NETWORK
TITLE = ---- Accion del Evento --> Peticion de Refresco del Dispositivo Barrera
///////////////////////////////////////////////////////////////////////////////
///////////////////////////////////////////////////////////////////////////////
///////////////////////////////////////////////////////////////////////////////
// Dispositivos tipo Barrera uno determinado o todos
DispositivoBarrera_EventoRecibido_RefrescoDispositivo:NOP   0;
      SET;
      L     #AtributosDeDispositivos.Numero;  // Mirar si hay numero de maquina
      L     0;  // Son todos las Barreras
      ==I;
      JC    DispositivosTodosBarrera_EventoRecibido_RefrescoDispositivo;


///////////////////////////////////////////////////////////////////////////////
// --- Es Una Maquina Determinada
      JU    DispositivosUnaBarrera_EventoRecibido_RefrescoDispositivo;



NETWORK
TITLE = ---- ---- De una Barrera
///////////////////////////////////////////////////////////////////////////////
///////////////////////////////////////////////////////////////////////////////
///////////////////////////////////////////////////////////////////////////////
// --- Una Barrera  determinada
DispositivosUnaBarrera_EventoRecibido_RefrescoDispositivo:NOP   0;

      L     #AtributosDeDispositivos.Numero;  // Ver que Barrera es
      L     "CTE_OffsetMesa";
      -I;
      T     #VarTempDispositivos.Numero;

      L     #VarTempDispositivos.Numero;  // Comprobar el numero de Barrera
      L     1;  // No menor de 1
      <I;  // No es correcto
      JC    Final_EventoRecibido_RefrescoDispositivo;
      L     #VarTempDispositivos.Numero;
      L     "CTE_MaxDispositivosBarrera";  // No meyor que el parametro
      >I;  // No es correcto
      JC    Final_EventoRecibido_RefrescoDispositivo;


///////////////////////////////////////////////////////////////////////////////
// --- Activar Refresco del Dispositivo
///////////////////////////////////////////////////////////////////////////////
// Activar Refresco del Dispositivo
      SET;
      S     "DB839_DispositivosVarios".DispoBarrera[#VarTempDispositivos.Numero].RefrescoDatos;


///////////////////////////////////////////////////////////////////////////////
// --- Finalizar
      JU    Final_EventoRecibido_RefrescoDispositivo;



NETWORK
TITLE = ---- ---- De Todas las Barreras
////////////////////////////////////////////////////////////////////////////
////////////////////////////////////////////////////////////////////////////
////////////////////////////////////////////////////////////////////////////
// --- Peticion de Todos los dispositivos BARRERA
DispositivosTodosBarrera_EventoRecibido_RefrescoDispositivo:NOP   0;
      L     1;
      T     #IndiceDispositivosVarios;


////////////////////////////////////////////////////////////////////////////
////////////////////////////////////////////////////////////////////////////
////////////////////////////////////////////////////////////////////////////
BucleBarrera_EventoRecibido_RefrescoDispositivo:NOP   0;


///////////////////////////////////////////////////////////////////////////////
// Activar Refresco del Dispositivo
      SET;
      S     "DB839_DispositivosVarios".DispoBarrera[#IndiceDispositivosVarios].RefrescoDatos;
////////////////////////////////////////////////////////////////////////////
      L     #IndiceDispositivosVarios;  // Siguiente Dispositivo
      L     1;
      +I;
      T     #IndiceDispositivosVarios;

      L     #IndiceDispositivosVarios;
      L     "CTE_MaxDispositivosBarrera";
      >I;  // Ha superado el maximo ??
      JC    FinBucleBarrera_EventoRecibido_RefrescoDispositivo;

      JU    BucleBarrera_EventoRecibido_RefrescoDispositivo;  // Continuar en el Bucle


////////////////////////////////////////////////////////////////////////////
////////////////////////////////////////////////////////////////////////////
////////////////////////////////////////////////////////////////////////////
FinBucleBarrera_EventoRecibido_RefrescoDispositivo:NOP   0;
      JU    Final_EventoRecibido_RefrescoDispositivo;


NETWORK
TITLE = ---- Accion del Evento --> Peticion de Refresco del Dispositivo Puerta
///////////////////////////////////////////////////////////////////////////////
///////////////////////////////////////////////////////////////////////////////
///////////////////////////////////////////////////////////////////////////////
// Dispositivos tipo Puerta uno determinado o todos
DispositivoPuerta_EventoRecibido_RefrescoDispositivo:NOP   0;
      SET;
      L     #AtributosDeDispositivos.Numero;  // Mirar si hay numero de maquina
      L     0;  // Son todos las Puertas
      ==I;
      JC    DispositivosTodosPuerta_EventoRecibido_RefrescoDispositivo;


///////////////////////////////////////////////////////////////////////////////
// --- Es Una Maquina Determinada
      JU    DispositivosUnaPuerta_EventoRecibido_RefrescoDispositivo;



NETWORK
TITLE = ---- ---- De una Puerta
///////////////////////////////////////////////////////////////////////////////
///////////////////////////////////////////////////////////////////////////////
///////////////////////////////////////////////////////////////////////////////
// --- Uan Puerta determinada
DispositivosUnaPuerta_EventoRecibido_RefrescoDispositivo:NOP   0;

      L     #AtributosDeDispositivos.Numero;  // Ver que Puerta es
      L     "CTE_OffsetMesa";
      -I;
      T     #VarTempDispositivos.Numero;

      L     #VarTempDispositivos.Numero;  // Comprobar el numero de Puerta
      L     1;  // No menor de 1
      <I;  // No es correcto
      JC    Final_EventoRecibido_RefrescoDispositivo;
      L     #VarTempDispositivos.Numero;
      L     "CTE_MaxDispositivosPuerta";  // No meyor que el parametro
      >I;  // No es correcto
      JC    Final_EventoRecibido_RefrescoDispositivo;


///////////////////////////////////////////////////////////////////////////////
// --- Activar Refresco del Dispositivo
///////////////////////////////////////////////////////////////////////////////
// Activar Refresco del Dispositivo
      SET;
      S     "DB839_DispositivosVarios".DispoPuerta[#VarTempDispositivos.Numero].RefrescoDatos;


///////////////////////////////////////////////////////////////////////////////
// --- Finalizar
      JU    Final_EventoRecibido_RefrescoDispositivo;



NETWORK
TITLE = ---- ---- De Todas las Puertas
////////////////////////////////////////////////////////////////////////////
////////////////////////////////////////////////////////////////////////////
////////////////////////////////////////////////////////////////////////////
// --- Peticion de Todos los dispositivos PUERTA
DispositivosTodosPuerta_EventoRecibido_RefrescoDispositivo:NOP   0;
      L     1;
      T     #IndiceDispositivosVarios;


////////////////////////////////////////////////////////////////////////////
////////////////////////////////////////////////////////////////////////////
////////////////////////////////////////////////////////////////////////////
BuclePuerta_EventoRecibido_RefrescoDispositivo:NOP   0;


///////////////////////////////////////////////////////////////////////////////
// Activar Refresco del Dispositivo
      SET;
      S     "DB839_DispositivosVarios".DispoPuerta[#IndiceDispositivosVarios].RefrescoDatos;

////////////////////////////////////////////////////////////////////////////
      L     #IndiceDispositivosVarios;  // Siguiente Dispositivo
      L     1;
      +I;
      T     #IndiceDispositivosVarios;

      L     #IndiceDispositivosVarios;
      L     "CTE_MaxDispositivosPuerta";
      >I;  // Ha superado el maximo ??
      JC    FinBuclePuerta_EventoRecibido_RefrescoDispositivo;

      JU    BuclePuerta_EventoRecibido_RefrescoDispositivo;  // Continuar en el Bucle


////////////////////////////////////////////////////////////////////////////
////////////////////////////////////////////////////////////////////////////
////////////////////////////////////////////////////////////////////////////
FinBuclePuerta_EventoRecibido_RefrescoDispositivo:NOP   0;
      JU    Final_EventoRecibido_RefrescoDispositivo;


NETWORK
TITLE = ---- Accion del Evento --> Peticion de Refresco del Dispositivo Linea de Potencia
///////////////////////////////////////////////////////////////////////////////
///////////////////////////////////////////////////////////////////////////////
///////////////////////////////////////////////////////////////////////////////
// Dispositivos tipo Linea de Potencia uno determinado o todos
DispositivoLineaPotencia_EventoRecibido_RefrescoDispositivo:NOP   0;
      SET;
      L     #AtributosDeDispositivos.Numero;  // Mirar si hay numero de maquina
      L     0;  // Son todos las Lineas de Potencia
      ==I;
      JC    DispositivosTodosLineaPotencia_EventoRecibido_RefrescoDispositivo;


///////////////////////////////////////////////////////////////////////////////
// --- Es Una Maquina Determinada
      JU    DispositivosUnaLineaPotencia_EventoRecibido_RefrescoDispositivo;



NETWORK
TITLE = ---- ---- De una Linea de Potencia
///////////////////////////////////////////////////////////////////////////////
///////////////////////////////////////////////////////////////////////////////
///////////////////////////////////////////////////////////////////////////////
// --- Maquina  determinada
DispositivosUnaLineaPotencia_EventoRecibido_RefrescoDispositivo:NOP   0;

      L     #AtributosDeDispositivos.Numero;  // Ver que Linea de Potencia es
      L     "CTE_OffsetMesa";
      -I;
      T     #VarTempDispositivos.Numero;

      L     #VarTempDispositivos.Numero;  // Comprobar el numero de Linea de Potencia
      L     1;  // No menor de 1
      <I;  // No es correcto
      JC    Final_EventoRecibido_RefrescoDispositivo;
      L     #VarTempDispositivos.Numero;
      L     "CTE_MaxDispositivosLineaPotencia";  // No meyor que el parametro
      >I;  // No es correcto
      JC    Final_EventoRecibido_RefrescoDispositivo;


///////////////////////////////////////////////////////////////////////////////
// --- Activar Refresco del Dispositivo
///////////////////////////////////////////////////////////////////////////////
// Activar Refresco del Dispositivo
      SET;
      S     "DB839_DispositivosVarios".DispoLineaPotencia[#VarTempDispositivos.Numero].RefrescoDatos;


///////////////////////////////////////////////////////////////////////////////
// --- Finalizar
      JU    Final_EventoRecibido_RefrescoDispositivo;



NETWORK
TITLE = ---- ---- De Todas Las Lineas de Potencia
////////////////////////////////////////////////////////////////////////////
////////////////////////////////////////////////////////////////////////////
////////////////////////////////////////////////////////////////////////////
// --- Peticion de Todos los dispositivos LINEA DE POTENCIA
DispositivosTodosLineaPotencia_EventoRecibido_RefrescoDispositivo:NOP   0;
      L     1;
      T     #IndiceDispositivosVarios;


////////////////////////////////////////////////////////////////////////////
////////////////////////////////////////////////////////////////////////////
////////////////////////////////////////////////////////////////////////////
BucleLineaPotencia_EventoRecibido_RefrescoDispositivo:NOP   0;


///////////////////////////////////////////////////////////////////////////////
// Activar Refresco del Dispositivo
      SET;
      S     "DB839_DispositivosVarios".DispoLineaPotencia[#IndiceDispositivosVarios].RefrescoDatos;

////////////////////////////////////////////////////////////////////////////
      L     #IndiceDispositivosVarios;  // Siguiente Dispositivo
      L     1;
      +I;
      T     #IndiceDispositivosVarios;

      L     #IndiceDispositivosVarios;
      L     "CTE_MaxDispositivosLineaPotencia";
      >I;  // Ha superado el maximo ??
      JC    FinBucleLineaPotencia_EventoRecibido_RefrescoDispositivo;

      JU    BucleLineaPotencia_EventoRecibido_RefrescoDispositivo;  // Continuar en el Bucle


////////////////////////////////////////////////////////////////////////////
////////////////////////////////////////////////////////////////////////////
////////////////////////////////////////////////////////////////////////////
FinBucleLineaPotencia_EventoRecibido_RefrescoDispositivo:NOP   0;
      JU    Final_EventoRecibido_RefrescoDispositivo;


NETWORK
TITLE = ---- Accion del Evento --> Peticion de Refresco de Todos Los Dispositivos
///////////////////////////////////////////////////////////////////////////////
///////////////////////////////////////////////////////////////////////////////
///////////////////////////////////////////////////////////////////////////////
// --- Todos los dispositivos
DispositivosTodos_EventoRecibido_RefrescoDispositivo:NOP   0;



NETWORK
TITLE = ---- ---- CCPIF y CBOX
///////////////////////////////////////////////////////////////////////////////
///////////////////////////////////////////////////////////////////////////////
///////////////////////////////////////////////////////////////////////////////
// --- Recorrer CCPIF y Todos los CBOX
      L     0;
      T     #IndiceCBOX;


///////////////////////////////////////////////////////////////////////////////
///////////////////////////////////////////////////////////////////////////////
///////////////////////////////////////////////////////////////////////////////
BucleArmarios_DispositivosTodos_EventoRecibido_RefrescoDispositivo:NOP   0;


///////////////////////////////////////////////////////////////////////////////
/// --- Inicio si pertenece al JDT
      SET;
      X     "DB855_DefinicionDispositivos".Dispositivos[#IndiceCBOX].EventosDelJdT02;
      XN    #JDT02_Activo;
      =     #DispositivoDeJDT02;

      SET;
      AN    #DispositivoDeJDT02;
      JC    ContinuarBucleArmarios_DispositivosTodos_EventoRecibido_RefrescoDispositivo;


///////////////////////////////////////////////////////////////////////////////
// --- Activar Refresco del Dispositivo
      L     250;  // 250 - Recibido Evento de Refresco de Datos del Dispositivo
      T     "DB830_Dispositivos".Dispositivos[#IndiceCBOX].EstadoRecepcionEvento;


///////////////////////////////////////////////////////////////////////////////
ContinuarBucleArmarios_DispositivosTodos_EventoRecibido_RefrescoDispositivo:NOP   0;
      L     #IndiceCBOX;  // Incremento al siguiente CBOX
      L     1;
      +I;
      T     #IndiceCBOX;

      L     #IndiceCBOX;
      L     "CTE_MaxDispositivos";
      >I;  // Finalizar
      JC    FinBucleArmarios_DispositivosTodos_EventoRecibido_RefrescoDispositivos;

///////////////////////////////////////////////////////////////////////////////
// --- Ir hacia el siguiente CBOX
      JU    BucleArmarios_DispositivosTodos_EventoRecibido_RefrescoDispositivo;


///////////////////////////////////////////////////////////////////////////////
///////////////////////////////////////////////////////////////////////////////
///////////////////////////////////////////////////////////////////////////////
FinBucleArmarios_DispositivosTodos_EventoRecibido_RefrescoDispositivos:NOP   0;



NETWORK
TITLE = ---- ---- Mesas
///////////////////////////////////////////////////////////////////////////////
///////////////////////////////////////////////////////////////////////////////
// Recorrer Todas las Mesas
      L     1;
      T     #IndiceMesa;

///////////////////////////////////////////////////////////////////////////////
///////////////////////////////////////////////////////////////////////////////
///////////////////////////////////////////////////////////////////////////////
BucleMesas_DispositivosTodos_EventoRecibido_RefrescoDispositivo:NOP   0;


///////////////////////////////////////////////////////////////////////////////
// --- Mirar si esta definido como mesa de Tracking y TL
      SET;
      AN    "DB850_DefinicionMesas".Mesa[#IndiceMesa].ConfigMesa.MesaPaso;
      AN    "DB850_DefinicionMesas".Mesa[#IndiceMesa].ConfigMesa.MesaCruce;
      AN    "DB850_DefinicionMesas".Mesa[#IndiceMesa].ConfigMesa.MesaMultiplesDestinos;
      AN    "DB850_DefinicionMesas".Mesa[#IndiceMesa].ConfigMesa.MesaTL;
      JC    ContinuarBucleMesas_DispositivosTodos_EventoRecibido_RefrescoDispositivo;


///////////////////////////////////////////////////////////////////////////////
// --- Mirar Si pertenece al JDT
      SET;
      X     "DB850_DefinicionMesas".Mesa[#IndiceMesa].ConfigMesa.MesaDeJDT02;  // JDT01 ?
      XN    #JDT02_Activo;
      =     #DispositivoDeJDT02;

      SET;
      AN    #DispositivoDeJDT02;
      JC    ContinuarBucleMesas_DispositivosTodos_EventoRecibido_RefrescoDispositivo;


///////////////////////////////////////////////////////////////////////////////
// --- Activar Refresco del Dispositivo
      L     250;  // 250 - Recibido Evento de Refresco de Datos del Dispositivo
      T     "DB831_Mesas".Mesas[#IndiceMesa].EstadoRecepcionEvento;


///////////////////////////////////////////////////////////////////////////////
ContinuarBucleMesas_DispositivosTodos_EventoRecibido_RefrescoDispositivo:NOP   0;

      L     #IndiceMesa;  // Incremento al siguiente Mesa
      L     1;
      +I;
      T     #IndiceMesa;

      L     #IndiceMesa;
      L     "CTE_MaxMesas";
      >I;  // Finalizar
      JC    FinBucleMesas_DispositivosTodos_EventoRecibido_RefrescoDispositivo;


///////////////////////////////////////////////////////////////////////////////
// --- Ir hacia el siguiente Mesa
      JU    BucleMesas_DispositivosTodos_EventoRecibido_RefrescoDispositivo;


///////////////////////////////////////////////////////////////////////////////
///////////////////////////////////////////////////////////////////////////////
///////////////////////////////////////////////////////////////////////////////
FinBucleMesas_DispositivosTodos_EventoRecibido_RefrescoDispositivo:NOP   0;



NETWORK
TITLE = ---- ---- Maquinas
///////////////////////////////////////////////////////////////////////////////
///////////////////////////////////////////////////////////////////////////////
///////////////////////////////////////////////////////////////////////////////
// Recorrer todas las Maquinas
      L     1;
      T     #IndiceMaquina;


///////////////////////////////////////////////////////////////////////////////
///////////////////////////////////////////////////////////////////////////////
///////////////////////////////////////////////////////////////////////////////
BucleMaquinas_DispositivosTodos_EventoRecibido_RefrescoDispositivo:NOP   0;


///////////////////////////////////////////////////////////////////////////////
// --- Mirar si esta definido como mesa de Tracking y TL
      SET;
      AN    "DB850_DefinicionMesas".Mesa[#IndiceMaquina].ConfigMesa.MesaPaso;
      AN    "DB850_DefinicionMesas".Mesa[#IndiceMaquina].ConfigMesa.MesaCruce;
      AN    "DB850_DefinicionMesas".Mesa[#IndiceMaquina].ConfigMesa.MesaMultiplesDestinos;
      AN    "DB850_DefinicionMesas".Mesa[#IndiceMaquina].ConfigMesa.MesaTL;
      JC    ContinuarBucleMaquinas_DispositivosTodos_EventoRecibido_RefrescoDispositivo;


///////////////////////////////////////////////////////////////////////////////
/// --- Mirar Si hay maquina
      SET;
      AN    "DB850_DefinicionMesas".Mesa[#IndiceMaquina].ConfigMesa.MaquinaEnMesa;  // Maquina ?
      JC    ContinuarBucleMaquinas_DispositivosTodos_EventoRecibido_RefrescoDispositivo;


///////////////////////////////////////////////////////////////////////////////
/// --- Mirar Si pertenece al JDT
      SET;
      X     "DB850_DefinicionMesas".Mesa[#IndiceMaquina].ConfigMesa.MesaDeJDT02;  // JDT01 ?
      XN    #JDT02_Activo;
      =     #MesaDeJDT02;

      SET;
      AN    #MesaDeJDT02;
      JC    ContinuarBucleMaquinas_DispositivosTodos_EventoRecibido_RefrescoDispositivo;


///////////////////////////////////////////////////////////////////////////////
// Activar Refresco del Dispositivo
      L     250;  // 250 - Recibido Evento de Refresco de Datos del Dispositivo
      T     "DB832_Maquinas".Maquinas[#IndiceMaquina].EstadoRecepcionEvento;


///////////////////////////////////////////////////////////////////////////////
ContinuarBucleMaquinas_DispositivosTodos_EventoRecibido_RefrescoDispositivo:NOP   0;
      L     #IndiceMaquina;  // Incremento al siguiente Maquina
      L     1;
      +I;
      T     #IndiceMaquina;

      L     #IndiceMaquina;
      L     "CTE_MaxMesas";
      >I;  // Finalizar
      JC    FinBucleMaquinas_DispositivosTodos_EventoRecibido_RefrescoDispositivo;


///////////////////////////////////////////////////////////////////////////////
// --- Ir hacia el siguiente Maquina
      JU    BucleMaquinas_DispositivosTodos_EventoRecibido_RefrescoDispositivo;


///////////////////////////////////////////////////////////////////////////////
///////////////////////////////////////////////////////////////////////////////
///////////////////////////////////////////////////////////////////////////////
FinBucleMaquinas_DispositivosTodos_EventoRecibido_RefrescoDispositivo:NOP   0;



NETWORK
TITLE = ---- ---- Balizas
////////////////////////////////////////////////////////////////////////////
////////////////////////////////////////////////////////////////////////////
////////////////////////////////////////////////////////////////////////////
// --- Peticion de Todos los dispositivos BALIZA

      L     1;
      T     #IndiceDispositivosVarios;


////////////////////////////////////////////////////////////////////////////
////////////////////////////////////////////////////////////////////////////
////////////////////////////////////////////////////////////////////////////
BucleBaliza_DispositivosTodos_EventoRecibido_RefrescoDispositivo:NOP   0;


///////////////////////////////////////////////////////////////////////////////
// Activar Refresco del Dispositivo
      SET;
      S     "DB839_DispositivosVarios".DispoBaliza[#IndiceDispositivosVarios].RefrescoDatos;
////////////////////////////////////////////////////////////////////////////
      L     #IndiceDispositivosVarios;  // Siguiente Dispositivo
      L     1;
      +I;
      T     #IndiceDispositivosVarios;

      L     #IndiceDispositivosVarios;
      L     "CTE_MaxDispositivosBaliza";
      >I;  // Ha superado el maximo ??
      JC    FinBucleBaliza_DispositivosTodos_EventoRecibido_RefrescoDispositivo;

      JU    BucleBaliza_DispositivosTodos_EventoRecibido_RefrescoDispositivo;  // Continuar en el Bucle


////////////////////////////////////////////////////////////////////////////
////////////////////////////////////////////////////////////////////////////
////////////////////////////////////////////////////////////////////////////
FinBucleBaliza_DispositivosTodos_EventoRecibido_RefrescoDispositivo:NOP   0;



NETWORK
TITLE = ---- ---- Llaves
////////////////////////////////////////////////////////////////////////////
////////////////////////////////////////////////////////////////////////////
////////////////////////////////////////////////////////////////////////////
// --- Peticion de Todos los dispositivos LLAVE

      L     1;
      T     #IndiceDispositivosVarios;


////////////////////////////////////////////////////////////////////////////
////////////////////////////////////////////////////////////////////////////
////////////////////////////////////////////////////////////////////////////
BucleLlave_DispositivosTodos_EventoRecibido_RefrescoDispositivo:NOP   0;


///////////////////////////////////////////////////////////////////////////////
// Activar Refresco del Dispositivo
      SET;
      S     "DB839_DispositivosVarios".DispoLlave[#IndiceDispositivosVarios].RefrescoDatos;
////////////////////////////////////////////////////////////////////////////
      L     #IndiceDispositivosVarios;  // Siguiente Dispositivo
      L     1;
      +I;
      T     #IndiceDispositivosVarios;

      L     #IndiceDispositivosVarios;
      L     "CTE_MaxDispositivosLlave";
      >I;  // Ha superado el maximo ??
      JC    FinBuclellave_DispositivosTodos_EventoRecibido_RefrescoDispositivo;

      JU    BucleLlave_DispositivosTodos_EventoRecibido_RefrescoDispositivo;  // Continuar en el Bucle


////////////////////////////////////////////////////////////////////////////
////////////////////////////////////////////////////////////////////////////
////////////////////////////////////////////////////////////////////////////
FinBuclellave_DispositivosTodos_EventoRecibido_RefrescoDispositivo:NOP   0;



NETWORK
TITLE = ---- ---- Setas
////////////////////////////////////////////////////////////////////////////
////////////////////////////////////////////////////////////////////////////
////////////////////////////////////////////////////////////////////////////
// --- Peticion de Todos los dispositivos SETA

      L     1;
      T     #IndiceDispositivosVarios;


////////////////////////////////////////////////////////////////////////////
////////////////////////////////////////////////////////////////////////////
////////////////////////////////////////////////////////////////////////////
BucleSeta_DispositivosTodos_EventoRecibido_RefrescoDispositivo:NOP   0;


///////////////////////////////////////////////////////////////////////////////
// Activar Refresco del Dispositivo
      SET;
      S     "DB839_DispositivosVarios".DispoSeta[#IndiceDispositivosVarios].RefrescoDatos;
////////////////////////////////////////////////////////////////////////////
      L     #IndiceDispositivosVarios;  // Siguiente Dispositivo
      L     1;
      +I;
      T     #IndiceDispositivosVarios;

      L     #IndiceDispositivosVarios;
      L     "CTE_MaxDispositivosSeta";
      >I;  // Ha superado el maximo ??
      JC    FinBucleSeta_DispositivosTodos_EventoRecibido_RefrescoDispositivo;

      JU    BucleSeta_DispositivosTodos_EventoRecibido_RefrescoDispositivo;  // Continuar en el Bucle


////////////////////////////////////////////////////////////////////////////
////////////////////////////////////////////////////////////////////////////
////////////////////////////////////////////////////////////////////////////
FinBucleSeta_DispositivosTodos_EventoRecibido_RefrescoDispositivo:NOP   0;



NETWORK
TITLE = ---- ---- Barreras
////////////////////////////////////////////////////////////////////////////
////////////////////////////////////////////////////////////////////////////
////////////////////////////////////////////////////////////////////////////
// --- Peticion de Todos los dispositivos BARRERA

      L     1;
      T     #IndiceDispositivosVarios;


////////////////////////////////////////////////////////////////////////////
////////////////////////////////////////////////////////////////////////////
////////////////////////////////////////////////////////////////////////////
BucleBarrera_DispositivosTodos_EventoRecibido_RefrescoDispositivo:NOP   0;


///////////////////////////////////////////////////////////////////////////////
// Activar Refresco del Dispositivo
      SET;
      S     "DB839_DispositivosVarios".DispoBarrera[#IndiceDispositivosVarios].RefrescoDatos;
////////////////////////////////////////////////////////////////////////////
      L     #IndiceDispositivosVarios;  // Siguiente Dispositivo
      L     1;
      +I;
      T     #IndiceDispositivosVarios;

      L     #IndiceDispositivosVarios;
      L     "CTE_MaxDispositivosBarrera";
      >I;  // Ha superado el maximo ??
      JC    FinBucleBarrera_DispositivosTodos_EventoRecibido_RefrescoDispositivo;

      JU    BucleBarrera_DispositivosTodos_EventoRecibido_RefrescoDispositivo;  // Continuar en el Bucle


////////////////////////////////////////////////////////////////////////////
////////////////////////////////////////////////////////////////////////////
////////////////////////////////////////////////////////////////////////////
FinBucleBarrera_DispositivosTodos_EventoRecibido_RefrescoDispositivo:NOP   0;



NETWORK
TITLE = ---- ---- Puertas
////////////////////////////////////////////////////////////////////////////
////////////////////////////////////////////////////////////////////////////
////////////////////////////////////////////////////////////////////////////
// --- Peticion de Todos los dispositivos PUERTA

      L     1;
      T     #IndiceDispositivosVarios;


////////////////////////////////////////////////////////////////////////////
////////////////////////////////////////////////////////////////////////////
////////////////////////////////////////////////////////////////////////////
BuclePuerta_DispositivosTodos_EventoRecibido_RefrescoDispositivo:NOP   0;


///////////////////////////////////////////////////////////////////////////////
// Activar Refresco del Dispositivo
      SET;
      S     "DB839_DispositivosVarios".DispoPuerta[#IndiceDispositivosVarios].RefrescoDatos;
////////////////////////////////////////////////////////////////////////////
      L     #IndiceDispositivosVarios;  // Siguiente Dispositivo
      L     1;
      +I;
      T     #IndiceDispositivosVarios;

      L     #IndiceDispositivosVarios;
      L     "CTE_MaxDispositivosPuerta";
      >I;  // Ha superado el maximo ??
      JC    FinBuclePuerta_DispositivosTodos_EventoRecibido_RefrescoDispositivo;

      JU    BuclePuerta_DispositivosTodos_EventoRecibido_RefrescoDispositivo;  // Continuar en el Bucle


////////////////////////////////////////////////////////////////////////////
////////////////////////////////////////////////////////////////////////////
////////////////////////////////////////////////////////////////////////////
FinBuclePuerta_DispositivosTodos_EventoRecibido_RefrescoDispositivo:NOP   0;



NETWORK
TITLE = ---- ---- Linea de Potencia
////////////////////////////////////////////////////////////////////////////
////////////////////////////////////////////////////////////////////////////
////////////////////////////////////////////////////////////////////////////
// --- Peticion de Todos los dispositivos LINEA DE POTENCIA

      L     1;
      T     #IndiceDispositivosVarios;


////////////////////////////////////////////////////////////////////////////
////////////////////////////////////////////////////////////////////////////
////////////////////////////////////////////////////////////////////////////
BucleLineaPotencia_DispositivosTodos_EventoRecibido_RefrescoDispositivo:NOP   0;


///////////////////////////////////////////////////////////////////////////////
// Activar Refresco del Dispositivo
      SET;
      S     "DB839_DispositivosVarios".DispoLineaPotencia[#IndiceDispositivosVarios].RefrescoDatos;
////////////////////////////////////////////////////////////////////////////
      L     #IndiceDispositivosVarios;  // Siguiente Dispositivo
      L     1;
      +I;
      T     #IndiceDispositivosVarios;

      L     #IndiceDispositivosVarios;
      L     "CTE_MaxDispositivosLineaPotencia";
      >I;  // Ha superado el maximo ??
      JC    FinBucleLineaPotencia_DispositivosTodos_EventoRecibido_RefrescoDispositivo;

      JU    BucleLineaPotencia_DispositivosTodos_EventoRecibido_RefrescoDispositivo;  // Continuar en el Bucle


////////////////////////////////////////////////////////////////////////////
////////////////////////////////////////////////////////////////////////////
////////////////////////////////////////////////////////////////////////////
FinBucleLineaPotencia_DispositivosTodos_EventoRecibido_RefrescoDispositivo:NOP   0;



NETWORK
TITLE = ---- Final
///////////////////////////////////////////////////////////////////////////////
///////////////////////////////////////////////////////////////////////////////
///////////////////////////////////////////////////////////////////////////////
// --- Se acabo el evento
Final_EventoRecibido_RefrescoDispositivo:NOP   0;
      L     #P_Eventos;  // Recupero por donde voy en la lista de eventos
      LAR2;  // Regreso a buscar el siguiente evento
      JU    FinBucle_EventosRecibidos;



NETWORK
TITLE = Evento DID0 - Notificacion de Cambio de Estado de Trabajo de un Dispositivo
// Analisis del evento
// - Inicializa variables de los atributos del Evento
// - Buscar Atributos o Final del Evento
// - Guardar datos del Evento
//   - Si es tipo CCPIF (50)
//   - Si es tipo CBOX (40)
//   - Si es tipo Mesa (60)
//   - Si es tipo Maquina (70)
// Analisis de los atributos de los eventos
// - Mirar que atributo del Evento es ?
// - Distribuir a recoger los datos del Evento
// - Recoger el Atributo Tipo de Dispositivo
// - Recoger el Atributo Numero de Dispositivo
// - Recoger el Atributo Nuevo Estado del Dispositivo
GuardarDatos_EventoRecibido_DIDO:NOP   0;

/////////////////////////////////////////////////////////////////////////
/////////////////////////////////////////////////////////////////////////
/////////////////////////////////////////////////////////////////////////
// --- Guardar Datos del Evento Recibido


/////////////////////////////////////////////////////////////////////////
/////////////////////////////////////////////////////////////////////////
/////////////////////////////////////////////////////////////////////////
/// --- Repartir segun tipo de dispositivo: CCPIF, CBOX, Mesa ...

      SET;  // Es CCPIF
      L     #AtributosDeDispositivos.Tipo;
      L     50;
      ==I;
      JC    DispositivoCCPIF_EventoRecibido_DIDO;

      SET;  // Es CBOX
      L     #AtributosDeDispositivos.Tipo;
      L     40;
      ==I;
      JC    DispositivoCBOX_EventoRecibido_DIDO;

      SET;  // Es Mesa
      L     #AtributosDeDispositivos.Tipo;
      L     60;
      ==I;
      JC    DispositivoMesa_EventoRecibido_DIDO;


/////////////////////////////////////////////////////////////////////////
/////////////////////////////////////////////////////////////////////////
/////////////////////////////////////////////////////////////////////////

      SET;  // Es VTDC
      L     #AtributosDeDispositivos.Tipo;
      L     "CTE_TipoMaquinaVTDC";
      ==I;
      JC    Dispositivo_VTDC_ELEV_EventoRecibido_DIDO;
      SET;  // Es ELEV
      L     #AtributosDeDispositivos.Tipo;
      L     "CTE_TipoMaquinaELEV";
      ==I;
      JC    Dispositivo_VTDC_ELEV_EventoRecibido_DIDO;

// Es Maquina 70 ... 99
      SET;
      A(;
      L     #AtributosDeDispositivos.Tipo;
      L     70;
      >=I;
      );
      A(;
      L     #AtributosDeDispositivos.Tipo;
      L     99;
      <=I;
      );
      JC    DispositivoMaquina_EventoRecibido_DIDO;


/////////////////////////////////////////////////////////////////////////
/////////////////////////////////////////////////////////////////////////
/////////////////////////////////////////////////////////////////////////
// No es ningun Tipo de Dispositivo esperado
      JU    Final_EventoRecibido_DIDO;



NETWORK
TITLE = ---- Accion del Evento --> Notificacion de Cambio de Estado de Trabajo del CCPIF
///////////////////////////////////////////////////////////////////////////////
///////////////////////////////////////////////////////////////////////////////
// --- Tipo CCPIF
DispositivoCCPIF_EventoRecibido_DIDO:NOP   0;
      L     #AtributosDeDispositivos.Numero;  // Comprobacion del numero de CCPIF
      L     "CTE_OffsetCCPIF";
      -I;
      L     1;
      <>I;  // Numero de CCPIF incorrecto
      JC    Final_EventoRecibido_DIDO;




// ????? -------------- ?????
// ????? Por ahora nada ?????
// ????? -------------- ?????




///////////////////////////////////////////////////////////////////////////////
// --- Finalizar
      JU    Final_EventoRecibido_DIDO;  // Finalizar



NETWORK
TITLE = ---- Accion del Evento --> Notificacion de Cambio de Estado de Trabajo del CBOX
///////////////////////////////////////////////////////////////////////////////
///////////////////////////////////////////////////////////////////////////////
// --- Tipo CBOX
DispositivoCBOX_EventoRecibido_DIDO:NOP   0;
      L     #AtributosDeDispositivos.Numero;  // Comprobacion del numero de CCPIF
      L     100;
      /I;
      L     "CTE_OffsetCCPIF";
      -I;
      L     1;
      <>I;  // Numero de CCPIF incorrecto
      JC    Final_EventoRecibido_DIDO;

      L     #AtributosDeDispositivos.Numero;  // Calculo del numero de CBOX
      L     100;
      MOD;  // Var verlo en la DB_Dispositivos
      T     #VarTempDispositivos.Numero;

      L     #VarTempDispositivos.Numero;  // Comprobacion del numero de CBOX
      L     1;  // Es menor de 1
      <I;  // No es correcto el numero de CBOX
      JC    Final_EventoRecibido_DIDO;
      L     #VarTempDispositivos.Numero;
      L     "CTE_MaxDispositivos";  // Si es mayor que el parametro
      >I;  // No es correcto el numero de CBOX
      JC    Final_EventoRecibido_DIDO;




// ????? -------------- ?????
// ????? Por ahora nada ?????
// ????? -------------- ?????




///////////////////////////////////////////////////////////////////////////////
// --- Finalizar
      JU    Final_EventoRecibido_DIDO;



NETWORK
TITLE = ---- Accion del Evento --> Notificacion de Cambio de Estado de Trabajo de la Mesa
///////////////////////////////////////////////////////////////////////////////
///////////////////////////////////////////////////////////////////////////////
// --- Tipo Mesa
DispositivoMesa_EventoRecibido_DIDO:NOP   0;
      L     #AtributosDeDispositivos.Numero;  // Ver que mesa es
      L     "CTE_OffsetMesa";
      -I;
      T     #VarTempDispositivos.Numero;

      L     #VarTempDispositivos.Numero;  // Comprobar el numero de mesa
      L     1;  // No menor de 1
      <I;  // No es correcto
      JC    Final_EventoRecibido_DIDO;
      L     #VarTempDispositivos.Numero;
      L     "CTE_MaxMesas";  // No meyor que el parametro
      >I;  // No es correcto
      JC    Final_EventoRecibido_DIDO;




// ????? -------------- ?????
// ????? Por ahora nada ?????
// ????? -------------- ?????




///////////////////////////////////////////////////////////////////////////////
// --- Finalizar
      JU    Final_EventoRecibido_DIDO;



NETWORK
TITLE = ---- Accion del Evento --> Notificacion de Cambio de Estado de Trabajo de la Maquina
///////////////////////////////////////////////////////////////////////////////
///////////////////////////////////////////////////////////////////////////////
// --- Tipo Maquina
DispositivoMaquina_EventoRecibido_DIDO:NOP   0;
      L     #AtributosDeDispositivos.Numero;  // Ver que mesa es
      L     "CTE_OffsetMesa";
      -I;
      T     #VarTempDispositivos.Numero;

      L     #VarTempDispositivos.Numero;  // Comprobar el numero de maquina
      L     1;  // No menor de 1
      <I;  // No es correcto
      JC    Final_EventoRecibido_DIDO;
      L     #VarTempDispositivos.Numero;
      L     "CTE_MaxMesas";  // No mayor que el parametro
      >I;  // No es correcto
      JC    Final_EventoRecibido_DIDO;


///////////////////////////////////////////////////////////////////////////////
// --- Comprobar si hay Orden a la Maquina

      L     #AtributosDeDispositivos.Operacion;
      L     0;
      ==I;
      JC    Final_EstadoTrabajoDeMaquina_EventoRecibido_DIDO;

///////////////////////////////////////////////////////////////////////////////
// ---Guardar Orden para la Maquina

      L     #AtributosDeDispositivos.Operacion;  // EstadoDispo + 0 ???
      L     0;  // Orden a guardar en el DB
      +I;
      T     "DB832_Maquinas".Maquinas[#VarTempDispositivos.Numero].Operacion;


///////////////////////////////////////////////////////////////////////////////
// --- Finalizar
Final_EstadoTrabajoDeMaquina_EventoRecibido_DIDO:NOP   0;
      JU    Final_EventoRecibido_DIDO;



NETWORK
TITLE = ---- Accion del Evento --> Notificacion de Cambio de Estado de Trabajo del VTDC / ELEV
///////////////////////////////////////////////////////////////////////////////
///////////////////////////////////////////////////////////////////////////////
// --- Tipo ELEV / VTDC
Dispositivo_VTDC_ELEV_EventoRecibido_DIDO:NOP   0;
      L     #AtributosDeDispositivos.Numero;  // Ver que mesa es
      L     "CTE_OffsetMesa";
      -I;
      T     #VarTempDispositivos.Numero;

      L     #VarTempDispositivos.Numero;  // Comprobacion del numero de VTDC
      L     1;  // Es menor de 1
      <I;  // No es correcto el numero de VTDC
      JC    Final_EventoRecibido_DIDO;
      L     #VarTempDispositivos.Numero;
      L     "CTE_MaxMesas";  // Si es mayor que el parametro
      >I;  // No es correcto el numero de VTDC
      JC    Final_EventoRecibido_DIDO;


///////////////////////////////////////////////////////////////////////////////
// --- Comprobar si hay Orden a la Maquina
      L     #AtributosDeDispositivos.Operacion;
      L     0;
      ==I;
      JC    Final_EstadoTrabajoDeVTDC_EventoRecibido_DIDO;


///////////////////////////////////////////////////////////////////////////////
// ---Guardar Orden para la Maquina
      L     #AtributosDeDispositivos.Operacion;  // EstadoDispo + 0 ???
      L     0;  // Orden a guardar en el DB
      +I;
      T     "DB832_Maquinas".Maquinas[#VarTempDispositivos.Numero].VTD_ELEV.Operacion;


///////////////////////////////////////////////////////////////////////////////
// --- Operacion >>> Orden del JDT de la Posicionar el VTD
      L     #AtributosDeDispositivos.Operacion;
      L     5001;
      <>I;  // --- Hay Orden ?
      JC    Final_EstadoTrabajoDeVTDC_EventoRecibido_DIDO;


      L     #AtributosDeDispositivos.MesaHorquilla;
      T     "DB832_Maquinas".Maquinas[#VarTempDispositivos.Numero].VTD_ELEV.MesaHorquilla;
      L     #AtributosDeDispositivos.MesaCargaDesCarga;
      T     "DB832_Maquinas".Maquinas[#VarTempDispositivos.Numero].VTD_ELEV.MesaCargaDesCarga;


///////////////////////////////////////////////////////////////////////////////
// --- Finalizar
Final_EstadoTrabajoDeVTDC_EventoRecibido_DIDO:NOP   0;
      JU    Final_EventoRecibido_DIDO;



NETWORK
TITLE = ---- Final
///////////////////////////////////////////////////////////////////////////////
///////////////////////////////////////////////////////////////////////////////
///////////////////////////////////////////////////////////////////////////////
// --- Se acabo el evento
Final_EventoRecibido_DIDO:NOP   0;
      L     #P_Eventos;  // Recupero por donde voy en la lista de eventos
      LAR2;  // Regreso a buscar el siguiente evento
      JU    FinBucle_EventosRecibidos;



NETWORK
TITLE = ////////////////////////////////////////////////////////////////////////////////////////////////////////////

NETWORK
TITLE = ----

NETWORK
TITLE = Tratamiento de los EVENTOS del ROUTER
// - Inicializa variables de los atributos del Evento
// - Buscar Atributos o Final del Evento
// - Guardar datos del Evento
// 
// Mirar que atributos del Evento es ?
// - Distribuir a recoger los datos del Evento
// - Recoger el Atributo Mckey
// - Recoger el Atributo Texto a Visualizar
/////////////////////////////////////////////////////////////////////////
/////////////////////////////////////////////////////////////////////////
/////////////////////////////////////////////////////////////////////////
EventosRecibidos_Router:NOP   0;

// -- Llamar a la funcion de tratamiento de Eventos del Router
      TAR2;
      T     #P_Eventos;  // Guardo, Por donde voy en la lista de eventos

//      CALL  "FC813_EventosRec_Router"
//         NumJdT         :=#NumJDT
//         PunteroEventos :=#P_Eventos

      CALL  "FC824_Recoge_Eventos_Routing"
      ( NumJdT          := #NumJDT,
        DBEventosrouter := "ROUT_DB_Eventos_Router",
        PunteroEventos  := #P_Eventos
      );


      L     #P_Eventos;  // Recupero, Por donde voy en la lista de eventos
      LAR2;

      JU    FinBucle_EventosRecibidos;



NETWORK
TITLE = Tratamiento de los EVENTOS del QUIMAROX
// - Inicializa variables de los atributos del Evento
// - Buscar Atributos o Final del Evento
// - Guardar datos del Evento
// 
// Mirar que atributos del Evento es ?
// - Distribuir a recoger los datos del Evento
// - Recoger el Atributo Mckey
// - Recoger el Atributo Texto a Visualizar
/////////////////////////////////////////////////////////////////////////
/////////////////////////////////////////////////////////////////////////
/////////////////////////////////////////////////////////////////////////
EventosRecibidos_Quimarox:NOP   0;

// -- Llamar a la funcion de tratamiento de Eventos del Router
      TAR2;
      T     #P_Eventos;  // Guardo, Por donde voy en la lista de eventos

      CALL  "FC605_EventosRec_Quimarox"
      ( NumJdT    := #NumJDT,
        P_Eventos := #P_Eventos
      );


      L     #P_Eventos;  // Recupero, Por donde voy en la lista de eventos
      LAR2;

      JU    FinBucle_EventosRecibidos;



NETWORK
TITLE = Tratamiento de los EVENTOS del RESET de V2
// - Inicializa variables de los atributos del Evento
// - Buscar Atributos o Final del Evento
// - Guardar datos del Evento
// 
// Mirar que atributos del Evento es ?
// - Distribuir a recoger los datos del Evento
// - Recoger el Atributo Mckey
// - Recoger el Atributo Texto a Visualizar
/////////////////////////////////////////////////////////////////////////
/////////////////////////////////////////////////////////////////////////
/////////////////////////////////////////////////////////////////////////
EventosRecibidos_Reset_V2:NOP   0;

// -- Llamar a la funcion de tratamiento de Eventos del Router
      TAR2;
      T     #P_Eventos;  // Guardo, Por donde voy en la lista de eventos

      CALL  "FC814_EventosRec_Reset"
      ( NumJdT    := #NumJDT,
        P_Eventos := #P_Eventos
      );


      L     #P_Eventos;  // Recupero, Por donde voy en la lista de eventos
      LAR2;

      JU    FinBucle_EventosRecibidos;



NETWORK
TITLE = Finalizar la Funcion
// Se acabo la función
/////////////////////////////////////////////////////////////////////////
/////////////////////////////////////////////////////////////////////////
/////////////////////////////////////////////////////////////////////////
FinalizarFuncion:NOP   0;


/////////////////////////////////////////////////////////////////////////
// Limpiar el DB del UltimoRecibido del JDT01
      L     #NumJDT;
      L     1;
      <>I;
      JC    NoLimpiarDB_JDT01;

      CALL  "FC898_BorrarMensaje"
      ( DB_A_RESET := "DB807_JDT01EventosRecibidos"
      );

NoLimpiarDB_JDT01:NOP   0;

/////////////////////////////////////////////////////////////////////////
// Limpiar el DB del UltimoRecibido del JDT01
      L     #NumJDT;
      L     2;
      <>I;
      JC    NoLimpiarDB_JDT02;

      CALL  "FC898_BorrarMensaje"
      ( DB_A_RESET := "DB708_JDT02EventosRecibidos"
      );

/////////////////////////////////////////////////////////////////////////
NoLimpiarDB_JDT02:NOP   0;


/////////////////////////////////////////////////////////////////////////
NoLimpiarNada:NOP   0;


END_FUNCTION
